TYPE Room_State_PassiveHeating_Hmi :
STRUCT
END_STRUCT
END_TYPE

(* stored: Version 1.1.0.1
   DUT Room_State_PassiveHeating_Hmi: Id {19942d14-7b9a-419a-9d53-abe959d99cdb} *)
